FUNCTION_BLOCK FB_Step
VAR_INPUT
	iNumber:INT; //requested number of the step
	iDepth:BOOL; //TRUE if the step has been completed to depth
END_VAR
VAR_OUTPUT
	qGo:BOOL; //TRUE to actuate the step
	qIsLastStep:BOOL; //TRUE if the step number is the last step
END_VAR
VAR
	tStepLive: BOOL;
	tSeqNotActive: BOOL;
	tNextNum: INT;
	j: INT;
	tNextStepNum: INT;
	osrDepth:R_TRIG;
END_VAR
VAR_IN_OUT
	stationState:typeStationMode;
END_VAR

//enable function
//IF stationState.AutoCycling OR TRUE THEN
IF stationState.AutoCycling OR TRUE THEN
	tStepLive := TRUE;
	ELSE
	tStepLive := FALSE;
END_IF

//find next step num, the next number in squence of the array, or the next highest number
IF tStepLive THEN
	actFindNextStep();
	ELSE
	//nowt
END_IF

//check if step squencer is not active
IF tStepLive THEN
	IF stationState.stepNum = 0 THEN
			tSeqNotActive := TRUE;
		ELSE
			tSeqNotActive := FALSE;
		END_IF
	
	ELSE
	tSeqNotActive := TRUE;
END_IF

//if the previous step number, stepNum, then perform the step
IF tStepLive THEN
	IF stationState.stepNum = iNumber THEN
			qGo := TRUE;
		ELSE
			qGo := FALSE;
		END_IF
	
	ELSE
	qGo := FALSE;
END_IF

//state the last step
IF tNextStepNum = stationState.sizeofStepListing THEN
		qIsLastStep := TRUE;
	ELSE
		qIsLastStep := FALSE;
END_IF


//depth trigger
osrDepth(CLK := iDepth);
IF osrDepth.Q THEN
	stationState.stepNum := tNextStepNum;
	
	//loop around on complete max
	IF stationState.stepNum = stationState.sizeofStepListing THEN
		stationState.stepNum := 0;
	END_IF
	
END_IF

ACTION actFindNextStep:
//assign location of step
stationState.stepNumListing[iNumber] := iNumber;

//assign last step, for continuity
stationState.stepNumListing[stationState.sizeofStepListing] := stationState.sizeofStepListing;


//search for next step number, starting from the input from the current step, 
FOR j := iNumber TO stationState.sizeofStepListing DO
	//
	//find the next highest number
	IF stationState.stepNumListing[j] > iNumber THEN
		tNextStepNum := j; 
		
		//no further steps found, assign max possible number
		IF j = stationState.sizeofStepListing THEN
			tNextStepNum := stationState.sizeofStepListing;
			EXIT;
		END_IF
		
		EXIT;
	END_IF
END_FOR
END_ACTION

END_FUNCTION_BLOCK

(* stored: Version 1.1.0.1, ProductVersion 3.1.4024.11
   POU FB_Step: Id {61a658dd-5a98-09d1-28da-afd0d5f9d3a6}, SpecialFunc None
   Action actFindNextStep: Id {2a97f42f-5167-0878-0a4e-4131435005a2} *)
